Yaskawa INFORM job: AAA.JBI

/JOB
//NAME AAA
//POS
///NPOS 236,0,236,0,0,0
///TOOL 9
///POSTYPE PULSE
///PULSE
C00000=32284,66241,-3799,47450,58446,-17967
C00001=32395,66278,-3767,47420,58477,-17972
C00002=32339,66010,-3916,47751,58289,-17892
C00003=32450,66047,-3885,47721,58320,-17897
C00004=32395,65782,-4034,48054,58134,-17816
C00005=32506,65819,-4005,48024,58165,-17821
C00006=32452,65556,-4153,48357,57980,-17738
C00007=32564,65592,-4126,48328,58011,-17744
C00008=32511,65331,-4273,48662,57828,-17659
C00009=32623,65368,-4247,48634,57858,-17664
C00010=32572,65109,-4394,48968,57677,-17578
C00011=32683,65145,-4370,48940,57707,-17583
C00012=32634,64889,-4516,49276,57527,-17495
C00013=32745,64925,-4494,49249,57558,-17501
C00014=32856,64961,-4471,49222,57588,-17507
C00015=32809,64706,-4619,49559,57410,-17416
C00016=32920,64742,-4598,49532,57440,-17422
C00017=32874,64490,-4745,49871,57263,-17330
C00018=32986,64526,-4726,49845,57293,-17336
C00019=32942,64276,-4873,50185,57119,-17242
C00020=33054,64311,-4855,50160,57149,-17248
C00021=33012,64064,-5001,50502,56976,-17152
C00022=33123,64099,-4986,50477,57006,-17158
C00023=33084,63854,-5132,50820,56836,-17060
C00024=33195,63889,-5118,50796,56865,-17066
C00025=33158,63646,-5263,51142,56697,-16966
C00026=33269,63680,-5251,51118,56726,-16972
C00027=33234,63440,-5397,51465,56560,-16869
C00028=33346,63474,-5387,51442,56589,-16875
C00029=33458,63509,-5376,51419,56618,-16881
C00030=33425,63271,-5523,51770,56454,-16777
C00031=33537,63305,-5515,51747,56483,-16783
C00032=33507,63069,-5662,52100,56321,-16676
C00033=33619,63103,-5655,52078,56350,-16682
C00034=33592,62869,-5803,52433,56191,-16572
C00035=33704,62903,-5798,52413,56219,-16578
C00036=33680,62671,-5945,52770,56063,-16466
C00037=33792,62705,-5942,52750,56091,-16472
C00038=33771,62475,-6090,53111,55937,-16358
C00039=33883,62509,-6089,53091,55964,-16364
C00040=33865,62282,-6237,53455,55813,-16247
C00041=33977,62315,-6238,53436,55840,-16253
C00042=33963,62090,-6386,53803,55691,-16133
C00043=34075,62123,-6389,53785,55719,-16139
C00044=34187,62156,-6392,53767,55746,-16145
C00045=34176,61933,-6543,54138,55599,-16023
C00046=34288,61966,-6547,54121,55627,-16029
C00047=34281,61745,-6699,54495,55482,-15903
C00048=34393,61777,-6706,54479,55510,-15909
C00049=34389,61559,-6859,54857,55368,-15781
C00050=34501,61591,-6867,54841,55395,-15787
C00051=34501,61374,-7021,55223,55255,-15657
C00052=34613,61406,-7032,55208,55282,-15662
C00053=34617,61191,-7187,55594,55145,-15529
C00054=34729,61224,-7199,55580,55171,-15535
C00055=34737,61010,-7355,55969,55036,-15399
C00056=34849,61043,-7370,55956,55063,-15404
C00057=34961,61075,-7384,55944,55090,-15410
C00058=34973,60863,-7544,56338,54957,-15271
C00059=35085,60895,-7560,56326,54983,-15276
C00060=35100,60685,-7722,56724,54852,-15135
C00061=35212,60717,-7740,56713,54878,-15140
C00062=35232,60509,-7903,57116,54749,-14996
C00063=35344,60541,-7923,57106,54775,-15001
C00064=35367,60334,-8089,57513,54648,-14854
C00065=35479,60366,-8111,57503,54674,-14859
C00066=35506,60160,-8278,57914,54548,-14710
C00067=35618,60192,-8302,57906,54574,-14714
C00068=35649,59988,-8472,58321,54450,-14563
C00069=35760,60020,-8498,58314,54475,-14567
C00070=35795,59816,-8670,58733,54352,-14414
C00071=35907,59849,-8697,58726,54378,-14418
C00072=36018,59882,-8724,58719,54403,-14422
C00073=36056,59679,-8902,59144,54281,-14266
C00074=36167,59712,-8930,59138,54306,-14271
C00075=36209,59510,-9110,59567,54184,-14112
C00076=36320,59543,-9141,59561,54210,-14116
C00077=36365,59342,-9323,59994,54088,-13956
C00078=36475,59375,-9355,59989,54113,-13960
C00079=36524,59174,-9541,60426,53991,-13798
C00080=36634,59208,-9574,60422,54016,-13802
C00081=36685,59008,-9763,60862,53894,-13639
C00082=36795,59042,-9798,60859,53919,-13642
C00083=36849,58842,-9990,61302,53796,-13478
C00084=36959,58876,-10027,61299,53821,-13481
C00085=37015,58676,-10222,61745,53698,-13315
C00086=37124,58711,-10260,61744,53723,-13318
C00087=37233,58747,-10297,61742,53748,-13322
C00088=37292,58547,-10497,62192,53622,-13155
C00089=37400,58583,-10536,62191,53647,-13158
C00090=37461,58383,-10740,62643,53520,-12990
C00091=37569,58420,-10779,62642,53545,-12993
C00092=37631,58219,-10986,63097,53417,-12824
C00093=37739,58257,-11027,63097,53441,-12827
C00094=37802,58056,-11238,63554,53310,-12658
C00095=37909,58094,-11279,63554,53335,-12661
C00096=37974,57892,-11493,64012,53201,-12492
C00097=38081,57931,-11536,64013,53226,-12494
C00098=38188,57969,-11578,64013,53250,-12497
C00099=38294,58008,-11620,64013,53275,-12500
C00100=38401,58047,-11661,64013,53300,-12502
C00101=38507,58086,-11702,64013,53325,-12505
C00102=38614,58126,-11743,64013,53350,-12508
C00103=38721,58166,-11783,64012,53375,-12510
C00104=38827,58206,-11823,64012,53400,-12513
C00105=38934,58246,-11862,64011,53425,-12515
C00106=39040,58287,-11901,64010,53451,-12518
C00107=39147,58328,-11940,64009,53476,-12520
C00108=39254,58369,-11978,64008,53502,-12523
C00109=39360,58410,-12016,64007,53528,-12526
C00110=39467,58452,-12054,64006,53553,-12528
C00111=39573,58494,-12091,64004,53579,-12531
C00112=39680,58536,-12127,64002,53605,-12533
C00113=39786,58578,-12164,64001,53632,-12536
C00114=39893,58621,-12200,63999,53658,-12538
C00115=39999,58664,-12235,63996,53684,-12541
C00116=40106,58707,-12270,63994,53711,-12543
C00117=40212,58751,-12305,63992,53737,-12545
C00118=40319,58794,-12340,63989,53764,-12548
C00119=40425,58838,-12373,63986,53791,-12550
C00120=40532,58882,-12407,63983,53818,-12553
C00121=40638,58927,-12440,63980,53845,-12555
C00122=40745,58972,-12473,63977,53872,-12558
C00123=40851,59017,-12505,63974,53900,-12560
C00124=40958,59062,-12537,63970,53927,-12562
C00125=41064,59107,-12569,63966,53954,-12565
C00126=41171,59153,-12600,63963,53982,-12567
C00127=41277,59199,-12631,63959,54010,-12569
C00128=41384,59245,-12662,63955,54038,-12572
C00129=41490,59291,-12692,63950,54066,-12574
C00130=41596,59338,-12721,63946,54094,-12576
C00131=41703,59385,-12751,63942,54122,-12579
C00132=41809,59432,-12780,63937,54150,-12581
C00133=41916,59479,-12808,63932,54179,-12583
C00134=42022,59527,-12837,63927,54207,-12585
C00135=42129,59574,-12865,63922,54236,-12588
C00136=42235,59622,-12892,63917,54265,-12590
C00137=42341,59670,-12919,63911,54293,-12592
C00138=42448,59719,-12946,63906,54322,-12594
C00139=42553,59768,-12973,63901,54351,-12596
C00140=42659,59817,-12999,63895,54381,-12598
C00141=42735,59578,-13215,64342,54202,-12445
C00142=42840,59629,-13241,64336,54232,-12447
C00143=42915,59389,-13458,64781,54050,-12295
C00144=43020,59442,-13484,64775,54080,-12296
C00145=43094,59202,-13702,65217,53894,-12146
C00146=43197,59256,-13728,65212,53924,-12148
C00147=43270,59015,-13946,65651,53733,-11999
C00148=43373,59071,-13972,65646,53764,-12000
C00149=43445,58830,-14191,66081,53569,-11854
C00150=43546,58888,-14216,66076,53600,-11855
C00151=43648,58946,-14241,66071,53630,-11856
C00152=43717,58706,-14461,66503,53432,-11711
C00153=43818,58765,-14485,66498,53463,-11712
C00154=43886,58524,-14706,66926,53259,-11569
C00155=43986,58585,-14730,66921,53291,-11570
C00156=44052,58344,-14951,67345,53083,-11430
C00157=44151,58407,-14974,67340,53115,-11430
C00158=44215,58164,-15196,67760,52903,-11293
C00159=44313,58229,-15219,67755,52934,-11293
C00160=44376,57985,-15442,68171,52718,-11158
C00161=44472,58052,-15463,68165,52750,-11158
C00162=44533,57807,-15687,68576,52529,-11026
C00163=44628,57875,-15708,68570,52561,-11026
C00164=44724,57944,-15728,68564,52594,-11026
C00165=44781,57700,-15952,68970,52368,-10896
C00166=44876,57770,-15971,68964,52401,-10896
C00167=44931,57525,-16196,69365,52171,-10768
C00168=45024,57597,-16214,69359,52205,-10768
C00169=45078,57351,-16439,69755,51970,-10644
C00170=45170,57424,-16457,69748,52004,-10643
C00171=45221,57178,-16682,70139,51765,-10522
C00172=45312,57253,-16699,70132,51799,-10521
C00173=45361,57005,-16925,70517,51556,-10403
C00174=45450,57082,-16940,70510,51590,-10402
C00175=45497,56833,-17167,70889,51342,-10287
C00176=45586,56912,-17182,70882,51377,-10285
C00177=45630,56661,-17409,71256,51126,-10173
C00178=45717,56742,-17422,71248,51161,-10172
C00179=45805,56823,-17435,71241,51196,-10170
C00180=45845,56573,-17662,71609,50941,-10061
C00181=45932,56656,-17674,71601,50976,-10059
C00182=45970,56405,-17901,71963,50717,-9953
C00183=46055,56489,-17912,71955,50753,-9951
C00184=46091,56237,-18139,72311,50490,-9848
C00185=46175,56324,-18149,72303,50526,-9846
C00186=46209,56071,-18377,72653,50259,-9745
C00187=46291,56159,-18385,72645,50296,-9743
C00188=46323,55905,-18614,72988,50025,-9645
C00189=46404,55995,-18621,72980,50063,-9643
C00190=46433,55740,-18850,73318,49788,-9548
C00191=46514,55832,-18855,73309,49826,-9546
C00192=46540,55576,-19085,73641,49548,-9454
C00193=46620,55669,-19089,73633,49587,-9452
C00194=46699,55763,-19093,73624,49625,-9449
C00195=46722,55508,-19322,73950,49345,-9360
C00196=46801,55603,-19325,73941,49384,-9357
C00197=46821,55348,-19554,74261,49100,-9271
C00198=46899,55445,-19555,74252,49139,-9268
C00199=46917,55189,-19785,74565,48852,-9184
C00200=46993,55288,-19785,74557,48892,-9181
C00201=47010,55031,-20015,74864,48602,-9100
C00202=47084,55131,-20014,74855,48643,-9097
C00203=47099,54875,-20244,75157,48350,-9018
C00204=47172,54977,-20241,75148,48391,-9015
C00205=47185,54719,-20471,75444,48096,-8939
C00206=47257,54823,-20468,75435,48137,-8935
C00207=47330,54927,-20464,75426,48179,-8932
C00208=47339,54671,-20693,75717,47882,-8858
C00209=47410,54776,-20688,75708,47923,-8854
C00210=47417,54520,-20917,75992,47624,-8784
C00211=47488,54627,-20911,75983,47666,-8780
C00212=47493,54371,-21141,76262,47364,-8711
C00213=47562,54479,-21133,76253,47407,-8707
C00214=47565,54223,-21363,76526,47103,-8641
C00215=47633,54333,-21353,76517,47146,-8636
C00216=47634,54077,-21583,76785,46840,-8573
C00217=47701,54189,-21573,76776,46884,-8568
C00218=47701,53932,-21803,77038,46576,-8507
C00219=47767,54046,-21791,77029,46620,-8502
C00220=47764,53790,-22022,77286,46310,-8443
C00221=47829,53905,-22008,77278,46355,-8438
C00222=47894,54020,-21995,77269,46400,-8432
C00223=47888,53766,-22224,77521,46089,-8375
C00224=47953,53883,-22209,77512,46134,-8370
C00225=47945,53629,-22439,77758,45821,-8315
C00226=48008,53747,-22423,77750,45867,-8309
C00227=47999,53493,-22652,77991,45553,-8256
C00228=48061,53613,-22635,77983,45599,-8250
C00229=48050,53360,-22864,78219,45284,-8200
C00230=48111,53482,-22846,78211,45330,-8193
C00231=48099,53229,-23075,78442,45014,-8145
C00232=48159,53352,-23055,78434,45060,-8138
C00233=48144,53100,-23284,78660,44743,-8091
C00234=48204,53225,-23263,78653,44790,-8084
C00235=48188,52974,-23492,78874,44471,-8040
EC00000=-139565,206517
EC00001=-139528,206529
EC00002=-138313,206331
EC00003=-138276,206341
EC00004=-137068,206134
EC00005=-137032,206143
EC00006=-135830,205927
EC00007=-135795,205935
EC00008=-134601,205710
EC00009=-134566,205717
EC00010=-133380,205483
EC00011=-133346,205488
EC00012=-132167,205245
EC00013=-132134,205249
EC00014=-132101,205254
EC00015=-130932,205000
EC00016=-130899,205003
EC00017=-129739,204740
EC00018=-129707,204742
EC00019=-128556,204470
EC00020=-128526,204471
EC00021=-127384,204190
EC00022=-127355,204189
EC00023=-126224,203900
EC00024=-126195,203898
EC00025=-125075,203600
EC00026=-125047,203597
EC00027=-123938,203290
EC00028=-123912,203286
EC00029=-123885,203282
EC00030=-122790,202966
EC00031=-122764,202960
EC00032=-121681,202636
EC00033=-121656,202630
EC00034=-120586,202299
EC00035=-120563,202291
EC00036=-119507,201953
EC00037=-119485,201944
EC00038=-118443,201599
EC00039=-118422,201589
EC00040=-117395,201239
EC00041=-117376,201227
EC00042=-116364,200872
EC00043=-116346,200860
EC00044=-116328,200848
EC00045=-115334,200487
EC00046=-115317,200473
EC00047=-114340,200109
EC00048=-114325,200095
EC00049=-113364,199728
EC00050=-113351,199713
EC00051=-112408,199344
EC00052=-112396,199328
EC00053=-111471,198959
EC00054=-111461,198943
EC00055=-110554,198573
EC00056=-110545,198557
EC00057=-110536,198540
EC00058=-109650,198172
EC00059=-109642,198155
EC00060=-108774,197789
EC00061=-108769,197772
EC00062=-107920,197411
EC00063=-107915,197393
EC00064=-107085,197038
EC00065=-107082,197020
EC00066=-106271,196671
EC00067=-106270,196653
EC00068=-105476,196313
EC00069=-105476,196295
EC00070=-104701,195964
EC00071=-104703,195947
EC00072=-104704,195930
EC00073=-103948,195609
EC00074=-103951,195593
EC00075=-103211,195285
EC00076=-103215,195269
EC00077=-102491,194974
EC00078=-102496,194959
EC00079=-101787,194678
EC00080=-101794,194665
EC00081=-101099,194399
EC00082=-101106,194386
EC00083=-100424,194138
EC00084=-100433,194126
EC00085=-99762,193895
EC00086=-99771,193884
EC00087=-99781,193874
EC00088=-99121,193662
EC00089=-99131,193654
EC00090=-98480,193461
EC00091=-98491,193453
EC00092=-97848,193280
EC00093=-97858,193275
EC00094=-97221,193121
EC00095=-97232,193117
EC00096=-96599,192984
EC00097=-96609,192982
EC00098=-96618,192980
EC00099=-96627,192979
EC00100=-96635,192977
EC00101=-96644,192976
EC00102=-96652,192975
EC00103=-96659,192975
EC00104=-96667,192974
EC00105=-96674,192974
EC00106=-96681,192974
EC00107=-96688,192973
EC00108=-96694,192974
EC00109=-96700,192974
EC00110=-96706,192974
EC00111=-96712,192974
EC00112=-96717,192975
EC00113=-96722,192975
EC00114=-96727,192976
EC00115=-96731,192976
EC00116=-96735,192977
EC00117=-96739,192977
EC00118=-96743,192978
EC00119=-96746,192979
EC00120=-96749,192979
EC00121=-96752,192979
EC00122=-96754,192980
EC00123=-96756,192980
EC00124=-96758,192980
EC00125=-96760,192981
EC00126=-96761,192981
EC00127=-96762,192980
EC00128=-96762,192980
EC00129=-96763,192980
EC00130=-96763,192979
EC00131=-96762,192979
EC00132=-96762,192978
EC00133=-96761,192977
EC00134=-96760,192975
EC00135=-96759,192974
EC00136=-96757,192972
EC00137=-96755,192970
EC00138=-96753,192968
EC00139=-96751,192965
EC00140=-96749,192963
EC00141=-96046,193100
EC00142=-96043,193099
EC00143=-95330,193255
EC00144=-95327,193255
EC00145=-94604,193429
EC00146=-94599,193430
EC00147=-93866,193621
EC00148=-93860,193623
EC00149=-93114,193831
EC00150=-93107,193834
EC00151=-93099,193836
EC00152=-92340,194062
EC00153=-92330,194065
EC00154=-91557,194306
EC00155=-91546,194311
EC00156=-90759,194566
EC00157=-90747,194571
EC00158=-89944,194839
EC00159=-89930,194846
EC00160=-89113,195127
EC00161=-89097,195134
EC00162=-88263,195427
EC00163=-88245,195434
EC00164=-88228,195441
EC00165=-87376,195746
EC00166=-87357,195753
EC00167=-86489,196068
EC00168=-86467,196076
EC00169=-85582,196400
EC00170=-85559,196408
EC00171=-84658,196741
EC00172=-84633,196749
EC00173=-83714,197088
EC00174=-83687,197097
EC00175=-82752,197443
EC00176=-82723,197452
EC00177=-81771,197803
EC00178=-81741,197812
EC00179=-81710,197820
EC00180=-80740,198176
EC00181=-80708,198184
EC00182=-79721,198545
EC00183=-79687,198553
EC00184=-78684,198917
EC00185=-78648,198924
EC00186=-77630,199291
EC00187=-77592,199298
EC00188=-76558,199666
EC00189=-76519,199673
EC00190=-75469,200043
EC00191=-75428,200049
EC00192=-74364,200419
EC00193=-74322,200425
EC00194=-74280,200430
EC00195=-73199,200800
EC00196=-73155,200805
EC00197=-72061,201175
EC00198=-72016,201178
EC00199=-70907,201548
EC00200=-70861,201551
EC00201=-69739,201919
EC00202=-69691,201921
EC00203=-68556,202287
EC00204=-68508,202289
EC00205=-67360,202652
EC00206=-67310,202653
EC00207=-67260,202653
EC00208=-66099,203015
EC00209=-66048,203014
EC00210=-64875,203373
EC00211=-64823,203371
EC00212=-63639,203727
EC00213=-63586,203724
EC00214=-62391,204077
EC00215=-62337,204073
EC00216=-61131,204422
EC00217=-61076,204418
EC00218=-59860,204763
EC00219=-59804,204758
EC00220=-58578,205099
EC00221=-58522,205093
EC00222=-58465,205086
EC00223=-57229,205423
EC00224=-57172,205415
EC00225=-55926,205748
EC00226=-55868,205739
EC00227=-54613,206068
EC00228=-54555,206058
EC00229=-53292,206382
EC00230=-53232,206371
EC00231=-51961,206691
EC00232=-51901,206679
EC00233=-50621,206995
EC00234=-50561,206982
EC00235=-49274,207293
//INST
///DATE 2023/03/09 16:54
///ATTR SC,RW
///GROUP1 RB2
///GROUP2 ST1
NOP
MOVL C00000 V=28.3 +MOVJ EC00000 VJ=28.3
MOVL C00001 V=28.3 +MOVJ EC00001 VJ=28.3
MOVL C00002 V=87.9 +MOVJ EC00002 VJ=87.9
MOVL C00003 V=28.3 +MOVJ EC00003 VJ=28.3
MOVL C00004 V=87.7 +MOVJ EC00004 VJ=87.7
MOVL C00005 V=28.4 +MOVJ EC00005 VJ=28.4
MOVL C00006 V=87.5 +MOVJ EC00006 VJ=87.5
MOVL C00007 V=28.4 +MOVJ EC00007 VJ=28.4
MOVL C00008 V=87.3 +MOVJ EC00008 VJ=87.3
MOVL C00009 V=28.4 +MOVJ EC00009 VJ=28.4
MOVL C00010 V=87.0 +MOVJ EC00010 VJ=87.0
MOVL C00011 V=28.4 +MOVJ EC00011 VJ=28.4
MOVL C00012 V=86.7 +MOVJ EC00012 VJ=86.7
MOVL C00013 V=28.5 +MOVJ EC00013 VJ=28.5
MOVL C00014 V=28.5 +MOVJ EC00014 VJ=28.5
MOVL C00015 V=86.4 +MOVJ EC00015 VJ=86.4
MOVL C00016 V=28.5 +MOVJ EC00016 VJ=28.5
MOVL C00017 V=86.1 +MOVJ EC00017 VJ=86.1
MOVL C00018 V=28.5 +MOVJ EC00018 VJ=28.5
MOVL C00019 V=85.7 +MOVJ EC00019 VJ=85.7
MOVL C00020 V=28.6 +MOVJ EC00020 VJ=28.6
MOVL C00021 V=85.3 +MOVJ EC00021 VJ=85.3
MOVL C00022 V=28.6 +MOVJ EC00022 VJ=28.6
MOVL C00023 V=84.9 +MOVJ EC00023 VJ=84.9
MOVL C00024 V=28.7 +MOVJ EC00024 VJ=28.7
MOVL C00025 V=84.4 +MOVJ EC00025 VJ=84.4
MOVL C00026 V=28.7 +MOVJ EC00026 VJ=28.7
MOVL C00027 V=83.9 +MOVJ EC00027 VJ=83.9
MOVL C00028 V=28.8 +MOVJ EC00028 VJ=28.8
MOVL C00029 V=28.8 +MOVJ EC00029 VJ=28.8
MOVL C00030 V=83.5 +MOVJ EC00030 VJ=83.5
MOVL C00031 V=28.8 +MOVJ EC00031 VJ=28.8
MOVL C00032 V=82.9 +MOVJ EC00032 VJ=82.9
MOVL C00033 V=28.9 +MOVJ EC00033 VJ=28.9
MOVL C00034 V=82.4 +MOVJ EC00034 VJ=82.4
MOVL C00035 V=28.9 +MOVJ EC00035 VJ=28.9
MOVL C00036 V=81.8 +MOVJ EC00036 VJ=81.8
MOVL C00037 V=29.0 +MOVJ EC00037 VJ=29.0
MOVL C00038 V=81.1 +MOVJ EC00038 VJ=81.1
MOVL C00039 V=29.0 +MOVJ EC00039 VJ=29.0
MOVL C00040 V=80.5 +MOVJ EC00040 VJ=80.5
MOVL C00041 V=29.1 +MOVJ EC00041 VJ=29.1
MOVL C00042 V=79.8 +MOVJ EC00042 VJ=79.8
MOVL C00043 V=29.2 +MOVJ EC00043 VJ=29.2
MOVL C00044 V=29.2 +MOVJ EC00044 VJ=29.2
MOVL C00045 V=79.2 +MOVJ EC00045 VJ=79.2
MOVL C00046 V=29.2 +MOVJ EC00046 VJ=29.2
MOVL C00047 V=78.5 +MOVJ EC00047 VJ=78.5
MOVL C00048 V=29.3 +MOVJ EC00048 VJ=29.3
MOVL C00049 V=77.8 +MOVJ EC00049 VJ=77.8
MOVL C00050 V=29.4 +MOVJ EC00050 VJ=29.4
MOVL C00051 V=77.0 +MOVJ EC00051 VJ=77.0
MOVL C00052 V=29.4 +MOVJ EC00052 VJ=29.4
MOVL C00053 V=76.3 +MOVJ EC00053 VJ=76.3
MOVL C00054 V=29.5 +MOVJ EC00054 VJ=29.5
MOVL C00055 V=75.5 +MOVJ EC00055 VJ=75.5
MOVL C00056 V=29.6 +MOVJ EC00056 VJ=29.6
MOVL C00057 V=29.6 +MOVJ EC00057 VJ=29.6
MOVL C00058 V=74.8 +MOVJ EC00058 VJ=74.8
MOVL C00059 V=29.7 +MOVJ EC00059 VJ=29.7
MOVL C00060 V=74.0 +MOVJ EC00060 VJ=74.0
MOVL C00061 V=29.7 +MOVJ EC00061 VJ=29.7
MOVL C00062 V=73.3 +MOVJ EC00062 VJ=73.3
MOVL C00063 V=29.8 +MOVJ EC00063 VJ=29.8
MOVL C00064 V=72.5 +MOVJ EC00064 VJ=72.5
MOVL C00065 V=29.9 +MOVJ EC00065 VJ=29.9
MOVL C00066 V=71.8 +MOVJ EC00066 VJ=71.8
MOVL C00067 V=29.9 +MOVJ EC00067 VJ=29.9
MOVL C00068 V=71.1 +MOVJ EC00068 VJ=71.1
MOVL C00069 V=30.0 +MOVJ EC00069 VJ=30.0
MOVL C00070 V=70.4 +MOVJ EC00070 VJ=70.4
MOVL C00071 V=30.1 +MOVJ EC00071 VJ=30.1
MOVL C00072 V=30.1 +MOVJ EC00072 VJ=30.1
MOVL C00073 V=69.8 +MOVJ EC00073 VJ=69.8
MOVL C00074 V=30.1 +MOVJ EC00074 VJ=30.1
MOVL C00075 V=69.2 +MOVJ EC00075 VJ=69.2
MOVL C00076 V=30.2 +MOVJ EC00076 VJ=30.2
MOVL C00077 V=68.6 +MOVJ EC00077 VJ=68.6
MOVL C00078 V=30.2 +MOVJ EC00078 VJ=30.2
MOVL C00079 V=68.1 +MOVJ EC00079 VJ=68.1
MOVL C00080 V=30.3 +MOVJ EC00080 VJ=30.3
MOVL C00081 V=67.6 +MOVJ EC00081 VJ=67.6
MOVL C00082 V=30.3 +MOVJ EC00082 VJ=30.3
MOVL C00083 V=67.2 +MOVJ EC00083 VJ=67.2
MOVL C00084 V=30.4 +MOVJ EC00084 VJ=30.4
MOVL C00085 V=66.8 +MOVJ EC00085 VJ=66.8
MOVL C00086 V=30.4 +MOVJ EC00086 VJ=30.4
MOVL C00087 V=30.4 +MOVJ EC00087 VJ=30.4
MOVL C00088 V=66.5 +MOVJ EC00088 VJ=66.5
MOVL C00089 V=30.4 +MOVJ EC00089 VJ=30.4
MOVL C00090 V=66.3 +MOVJ EC00090 VJ=66.3
MOVL C00091 V=30.4 +MOVJ EC00091 VJ=30.4
MOVL C00092 V=66.0 +MOVJ EC00092 VJ=66.0
MOVL C00093 V=30.5 +MOVJ EC00093 VJ=30.5
MOVL C00094 V=65.9 +MOVJ EC00094 VJ=65.9
MOVL C00095 V=30.5 +MOVJ EC00095 VJ=30.5
MOVL C00096 V=65.8 +MOVJ EC00096 VJ=65.8
MOVL C00097 V=30.4 +MOVJ EC00097 VJ=30.4
MOVL C00098 V=30.4 +MOVJ EC00098 VJ=30.4
MOVL C00099 V=30.4 +MOVJ EC00099 VJ=30.4
MOVL C00100 V=30.4 +MOVJ EC00100 VJ=30.4
MOVL C00101 V=30.4 +MOVJ EC00101 VJ=30.4
MOVL C00102 V=30.3 +MOVJ EC00102 VJ=30.3
MOVL C00103 V=30.3 +MOVJ EC00103 VJ=30.3
MOVL C00104 V=30.3 +MOVJ EC00104 VJ=30.3
MOVL C00105 V=30.3 +MOVJ EC00105 VJ=30.3
MOVL C00106 V=30.3 +MOVJ EC00106 VJ=30.3
MOVL C00107 V=30.3 +MOVJ EC00107 VJ=30.3
MOVL C00108 V=30.3 +MOVJ EC00108 VJ=30.3
MOVL C00109 V=30.3 +MOVJ EC00109 VJ=30.3
MOVL C00110 V=30.3 +MOVJ EC00110 VJ=30.3
MOVL C00111 V=30.2 +MOVJ EC00111 VJ=30.2
MOVL C00112 V=30.2 +MOVJ EC00112 VJ=30.2
MOVL C00113 V=30.2 +MOVJ EC00113 VJ=30.2
MOVL C00114 V=30.2 +MOVJ EC00114 VJ=30.2
MOVL C00115 V=30.2 +MOVJ EC00115 VJ=30.2
MOVL C00116 V=30.2 +MOVJ EC00116 VJ=30.2
MOVL C00117 V=30.2 +MOVJ EC00117 VJ=30.2
MOVL C00118 V=30.2 +MOVJ EC00118 VJ=30.2
MOVL C00119 V=30.1 +MOVJ EC00119 VJ=30.1
MOVL C00120 V=30.1 +MOVJ EC00120 VJ=30.1
MOVL C00121 V=30.1 +MOVJ EC00121 VJ=30.1
MOVL C00122 V=30.1 +MOVJ EC00122 VJ=30.1
MOVL C00123 V=30.1 +MOVJ EC00123 VJ=30.1
MOVL C00124 V=30.1 +MOVJ EC00124 VJ=30.1
MOVL C00125 V=30.1 +MOVJ EC00125 VJ=30.1
MOVL C00126 V=30.1 +MOVJ EC00126 VJ=30.1
MOVL C00127 V=30.0 +MOVJ EC00127 VJ=30.0
MOVL C00128 V=30.0 +MOVJ EC00128 VJ=30.0
MOVL C00129 V=30.0 +MOVJ EC00129 VJ=30.0
MOVL C00130 V=30.0 +MOVJ EC00130 VJ=30.0
MOVL C00131 V=30.0 +MOVJ EC00131 VJ=30.0
MOVL C00132 V=30.0 +MOVJ EC00132 VJ=30.0
MOVL C00133 V=30.0 +MOVJ EC00133 VJ=30.0
MOVL C00134 V=30.0 +MOVJ EC00134 VJ=30.0
MOVL C00135 V=29.9 +MOVJ EC00135 VJ=29.9
MOVL C00136 V=29.9 +MOVJ EC00136 VJ=29.9
MOVL C00137 V=29.9 +MOVJ EC00137 VJ=29.9
MOVL C00138 V=29.9 +MOVJ EC00138 VJ=29.9
MOVL C00139 V=29.9 +MOVJ EC00139 VJ=29.9
MOVL C00140 V=29.9 +MOVJ EC00140 VJ=29.9
MOVL C00141 V=68.7 +MOVJ EC00141 VJ=68.7
MOVL C00142 V=29.9 +MOVJ EC00142 VJ=29.9
MOVL C00143 V=68.9 +MOVJ EC00143 VJ=68.9
MOVL C00144 V=29.8 +MOVJ EC00144 VJ=29.8
MOVL C00145 V=69.2 +MOVJ EC00145 VJ=69.2
MOVL C00146 V=29.8 +MOVJ EC00146 VJ=29.8
MOVL C00147 V=69.6 +MOVJ EC00147 VJ=69.6
MOVL C00148 V=29.7 +MOVJ EC00148 VJ=29.7
MOVL C00149 V=70.0 +MOVJ EC00149 VJ=70.0
MOVL C00150 V=29.7 +MOVJ EC00150 VJ=29.7
MOVL C00151 V=29.7 +MOVJ EC00151 VJ=29.7
MOVL C00152 V=70.3 +MOVJ EC00152 VJ=70.3
MOVL C00153 V=29.6 +MOVJ EC00153 VJ=29.6
MOVL C00154 V=70.7 +MOVJ EC00154 VJ=70.7
MOVL C00155 V=29.5 +MOVJ EC00155 VJ=29.5
MOVL C00156 V=71.2 +MOVJ EC00156 VJ=71.2
MOVL C00157 V=29.4 +MOVJ EC00157 VJ=29.4
MOVL C00158 V=71.7 +MOVJ EC00158 VJ=71.7
MOVL C00159 V=29.4 +MOVJ EC00159 VJ=29.4
MOVL C00160 V=72.2 +MOVJ EC00160 VJ=72.2
MOVL C00161 V=29.3 +MOVJ EC00161 VJ=29.3
MOVL C00162 V=72.7 +MOVJ EC00162 VJ=72.7
MOVL C00163 V=29.2 +MOVJ EC00163 VJ=29.2
MOVL C00164 V=29.2 +MOVJ EC00164 VJ=29.2
MOVL C00165 V=73.2 +MOVJ EC00165 VJ=73.2
MOVL C00166 V=29.1 +MOVJ EC00166 VJ=29.1
MOVL C00167 V=73.8 +MOVJ EC00167 VJ=73.8
MOVL C00168 V=29.0 +MOVJ EC00168 VJ=29.0
MOVL C00169 V=74.3 +MOVJ EC00169 VJ=74.3
MOVL C00170 V=29.0 +MOVJ EC00170 VJ=29.0
MOVL C00171 V=74.9 +MOVJ EC00171 VJ=74.9
MOVL C00172 V=28.9 +MOVJ EC00172 VJ=28.9
MOVL C00173 V=75.5 +MOVJ EC00173 VJ=75.5
MOVL C00174 V=28.8 +MOVJ EC00174 VJ=28.8
MOVL C00175 V=76.1 +MOVJ EC00175 VJ=76.1
MOVL C00176 V=28.7 +MOVJ EC00176 VJ=28.7
MOVL C00177 V=76.7 +MOVJ EC00177 VJ=76.7
MOVL C00178 V=28.6 +MOVJ EC00178 VJ=28.6
MOVL C00179 V=28.6 +MOVJ EC00179 VJ=28.6
MOVL C00180 V=77.2 +MOVJ EC00180 VJ=77.2
MOVL C00181 V=28.5 +MOVJ EC00181 VJ=28.5
MOVL C00182 V=77.8 +MOVJ EC00182 VJ=77.8
MOVL C00183 V=28.4 +MOVJ EC00183 VJ=28.4
MOVL C00184 V=78.4 +MOVJ EC00184 VJ=78.4
MOVL C00185 V=28.4 +MOVJ EC00185 VJ=28.4
MOVL C00186 V=79.0 +MOVJ EC00186 VJ=79.0
MOVL C00187 V=28.3 +MOVJ EC00187 VJ=28.3
MOVL C00188 V=79.5 +MOVJ EC00188 VJ=79.5
MOVL C00189 V=28.2 +MOVJ EC00189 VJ=28.2
MOVL C00190 V=80.1 +MOVJ EC00190 VJ=80.1
MOVL C00191 V=28.1 +MOVJ EC00191 VJ=28.1
MOVL C00192 V=80.6 +MOVJ EC00192 VJ=80.6
MOVL C00193 V=28.1 +MOVJ EC00193 VJ=28.1
MOVL C00194 V=28.1 +MOVJ EC00194 VJ=28.1
MOVL C00195 V=81.1 +MOVJ EC00195 VJ=81.1
MOVL C00196 V=28.0 +MOVJ EC00196 VJ=28.0
MOVL C00197 V=81.6 +MOVJ EC00197 VJ=81.6
MOVL C00198 V=27.9 +MOVJ EC00198 VJ=27.9
MOVL C00199 V=82.1 +MOVJ EC00199 VJ=82.1
MOVL C00200 V=27.9 +MOVJ EC00200 VJ=27.9
MOVL C00201 V=82.6 +MOVJ EC00201 VJ=82.6
MOVL C00202 V=27.8 +MOVJ EC00202 VJ=27.8
MOVL C00203 V=83.1 +MOVJ EC00203 VJ=83.1
MOVL C00204 V=27.8 +MOVJ EC00204 VJ=27.8
MOVL C00205 V=83.6 +MOVJ EC00205 VJ=83.6
MOVL C00206 V=27.7 +MOVJ EC00206 VJ=27.7
MOVL C00207 V=27.7 +MOVJ EC00207 VJ=27.7
MOVL C00208 V=84.0 +MOVJ EC00208 VJ=84.0
MOVL C00209 V=27.7 +MOVJ EC00209 VJ=27.7
MOVL C00210 V=84.4 +MOVJ EC00210 VJ=84.4
MOVL C00211 V=27.6 +MOVJ EC00211 VJ=27.6
MOVL C00212 V=84.8 +MOVJ EC00212 VJ=84.8
MOVL C00213 V=27.6 +MOVJ EC00213 VJ=27.6
MOVL C00214 V=85.2 +MOVJ EC00214 VJ=85.2
MOVL C00215 V=27.5 +MOVJ EC00215 VJ=27.5
MOVL C00216 V=85.6 +MOVJ EC00216 VJ=85.6
MOVL C00217 V=27.5 +MOVJ EC00217 VJ=27.5
MOVL C00218 V=86.0 +MOVJ EC00218 VJ=86.0
MOVL C00219 V=27.4 +MOVJ EC00219 VJ=27.4
MOVL C00220 V=86.3 +MOVJ EC00220 VJ=86.3
MOVL C00221 V=27.4 +MOVJ EC00221 VJ=27.4
MOVL C00222 V=27.4 +MOVJ EC00222 VJ=27.4
MOVL C00223 V=86.6 +MOVJ EC00223 VJ=86.6
MOVL C00224 V=27.4 +MOVJ EC00224 VJ=27.4
MOVL C00225 V=87.0 +MOVJ EC00225 VJ=87.0
MOVL C00226 V=27.4 +MOVJ EC00226 VJ=27.4
MOVL C00227 V=87.3 +MOVJ EC00227 VJ=87.3
MOVL C00228 V=27.3 +MOVJ EC00228 VJ=27.3
MOVL C00229 V=87.6 +MOVJ EC00229 VJ=87.6
MOVL C00230 V=27.3 +MOVJ EC00230 VJ=27.3
MOVL C00231 V=87.8 +MOVJ EC00231 VJ=87.8
MOVL C00232 V=27.3 +MOVJ EC00232 VJ=27.3
MOVL C00233 V=88.1 +MOVJ EC00233 VJ=88.1
MOVL C00234 V=27.3 +MOVJ EC00234 VJ=27.3
MOVL C00235 V=88.3 +MOVJ EC00235 VJ=88.3
END
